(* Schneider Machine Expert - Basic project Seren_Alarm, file version 3.0.0.0 *)

HARDWARE
  Cpu 0: TM221CE16R
  EthernetConfiguration: NetworkName=M221, IpAllocationMode=FixedAddress, IpAddress=192.168.0.221, SubnetMask=255.255.255.0
  SerialLineConfiguration: Baud=Baud19200, Parity=ParityEven, DataBits=DataBits8, StopBits=StopBits1, PhysicalMedium=PhysicalMediumRs485, TransmissionMode=TransmissionModeModbusRtu, SlaveId=1, Addressing=SlaveAddressing
  MastTask: UsePeriodScanMode=false, PeriodScan=100
  FastTask: Period=255
  CpuBehavior: StartingMode=StartInRun, AutoSaveRamOnEeprom=true, WatchdogPeriod=250

SYMBOLS  (address, symbol, comment, settings)
  %M0       M_COM_OK
  %M1       M_HB_LAST
  %M2       M_HB_TOGGLED
  %M10      M_ENABLE_GEN
  %M11      M_PULSE_OUT
  %M12      M_PAUSE_OUT
  %M13      M_SERIES_PAUSE
  %S0       SB_COLDSTART  "Indicates or executes a cold start (data initialized to default values)"
  %MW0      PLC_CONTROL_WORD
  %MW1      PLC_STATUS_WORD
  %MW2      SOUND_PROFILE_CODE
  %MW3      SOUND_PULSE_COUNT
  %MW4      SOUND_PULSE_TIME_MS
  %MW5      SOUND_PAUSE_TIME_MS
  %MW6      SOUND_SERIES_INTERVAL_MS
  %MW10     ACTIVE_PULSE_COUNT
  %MW11     ACTIVE_PULSE_T_PRESET
  %MW12     ACTIVE_PAUSE_T_PRESET
  %MW13     ACTIVE_SERIES_T_PRESET
  %MW14     SERIES_COUNTER_VAL
  %TM0        [Preset=12, Base=OneSecond]
  %TM1        [Preset=2, Base=OneHundredMilliSeconds]
  %TM2        [Preset=3, Base=OneHundredMilliSeconds]
  %TM3        [Preset=30, Base=OneSecond]
  %QWM0     QW_HEARD_BEAT_WORD
  %QWM1     QW_PLC_CONTROL_WORD
  %IWM0     IW_PLC_HEARD_BEAT_WORD
  %IWM1     IW_PLC_STATUS_WORD

POU SIREN_CONTROL
  (* SectionNumber=1 *)

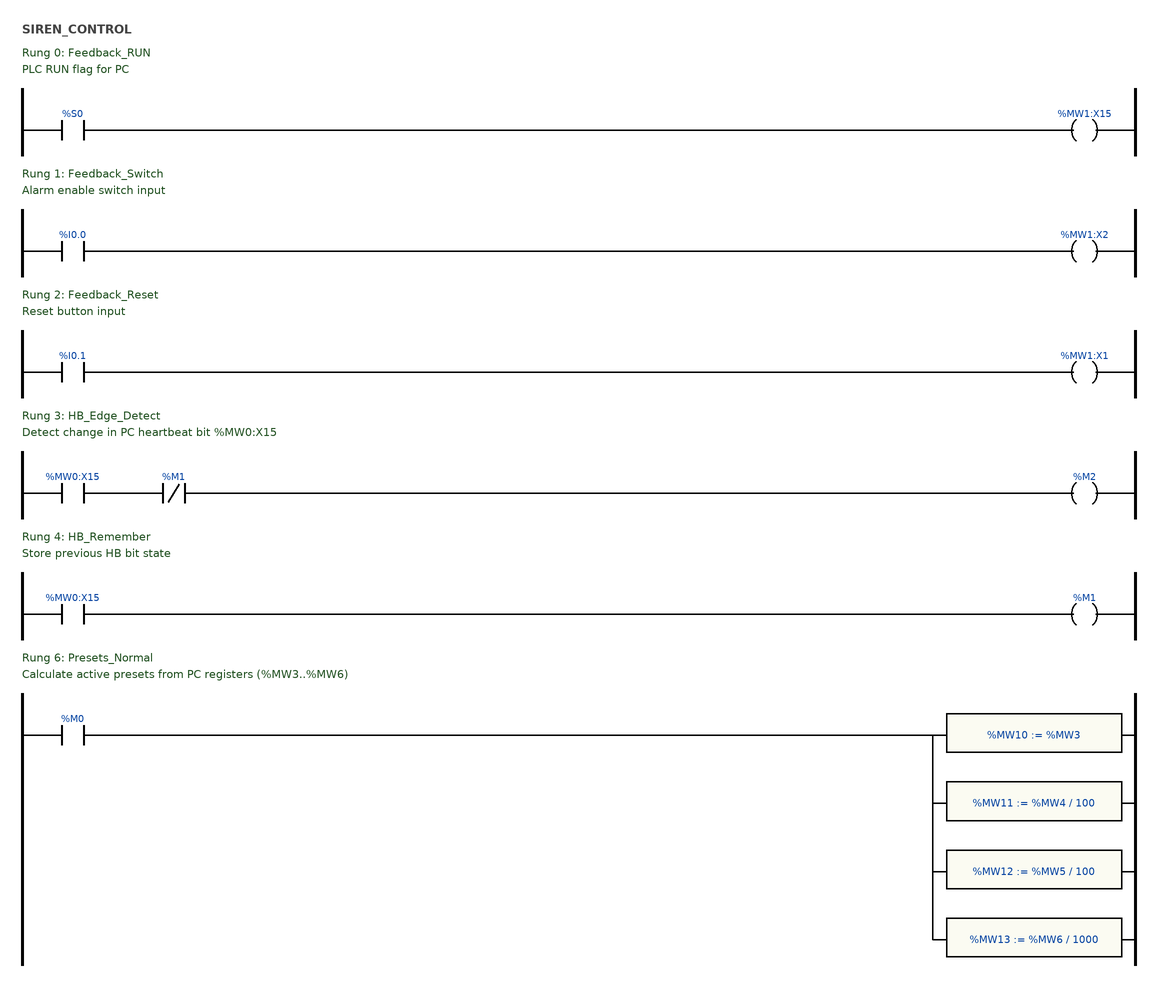

// Rung 0: Feedback_RUN
// PLC RUN flag for PC
  LD %S0                  (* SB_COLDSTART *)
  ST %MW1:X15             (* PLC_STATUS_WORD *)
  // as ST:
  //   PLC_STATUS_WORD:X15 := SB_COLDSTART;

// Rung 1: Feedback_Switch
// Alarm enable switch input
  LD %I0.0
  ST %MW1:X2              (* PLC_STATUS_WORD *)
  // as ST:
  //   PLC_STATUS_WORD:X2 := %I0.0;

// Rung 2: Feedback_Reset
// Reset button input
  LD %I0.1
  ST %MW1:X1              (* PLC_STATUS_WORD *)
  // as ST:
  //   PLC_STATUS_WORD:X1 := %I0.1;

// Rung 3: HB_Edge_Detect
// Detect change in PC heartbeat bit %MW0:X15
  LD %MW0:X15             (* PLC_CONTROL_WORD *)
  ANDN %M1                (* M_HB_LAST *)
  ST %M2                  (* M_HB_TOGGLED *)
  // as ST:
  //   M_HB_TOGGLED := PLC_CONTROL_WORD:X15 AND NOT M_HB_LAST;

// Rung 4: HB_Remember
// Store previous HB bit state
  LD %MW0:X15             (* PLC_CONTROL_WORD *)
  ST %M1                  (* M_HB_LAST *)
  // as ST:
  //   M_HB_LAST := PLC_CONTROL_WORD:X15;

// Rung 5: Watchdog_Timer
// Watchdog: %M0 is 1 while communication is OK, 0 when lost
  BLK %TM0
  LDN %M2                 (* M_HB_TOGGLED *)
  IN
  OUT_BLK
  LDN Q
  ST %M0                  (* M_COM_OK *)
  END_BLK
  // as ST:
  //   %TM0(IN := NOT M_HB_TOGGLED);
  //   M_COM_OK := NOT %TM0.Q;
  (* the ladder stored for this rung does not match its IL; not drawn *)

// Rung 6: Presets_Normal
// Calculate active presets from PC registers (%MW3..%MW6)
  LD %M0                  (* M_COM_OK *)
  [ %MW10 := %MW3 ]       (* ACTIVE_PULSE_COUNT, SOUND_PULSE_COUNT *)
  [ %MW11 := %MW4 / 100 ] (* ACTIVE_PULSE_T_PRESET, SOUND_PULSE_TIME_MS *)
  [ %MW12 := %MW5 / 100 ] (* ACTIVE_PAUSE_T_PRESET, SOUND_PAUSE_TIME_MS *)
  [ %MW13 := %MW6 / 1000 ](* ACTIVE_SERIES_T_PRESET, SOUND_SERIES_INTERVAL_MS *)
  // as ST:
  //   IF M_COM_OK THEN ACTIVE_PULSE_COUNT := SOUND_PULSE_COUNT; END_IF;
  //   IF M_COM_OK THEN ACTIVE_PULSE_T_PRESET := SOUND_PULSE_TIME_MS / 100; END_IF;
  //   IF M_COM_OK THEN ACTIVE_PAUSE_T_PRESET := SOUND_PAUSE_TIME_MS / 100; END_IF;
  //   IF M_COM_OK THEN ACTIVE_SERIES_T_PRESET := SOUND_SERIES_INTERVAL_MS / 1000; END_IF;

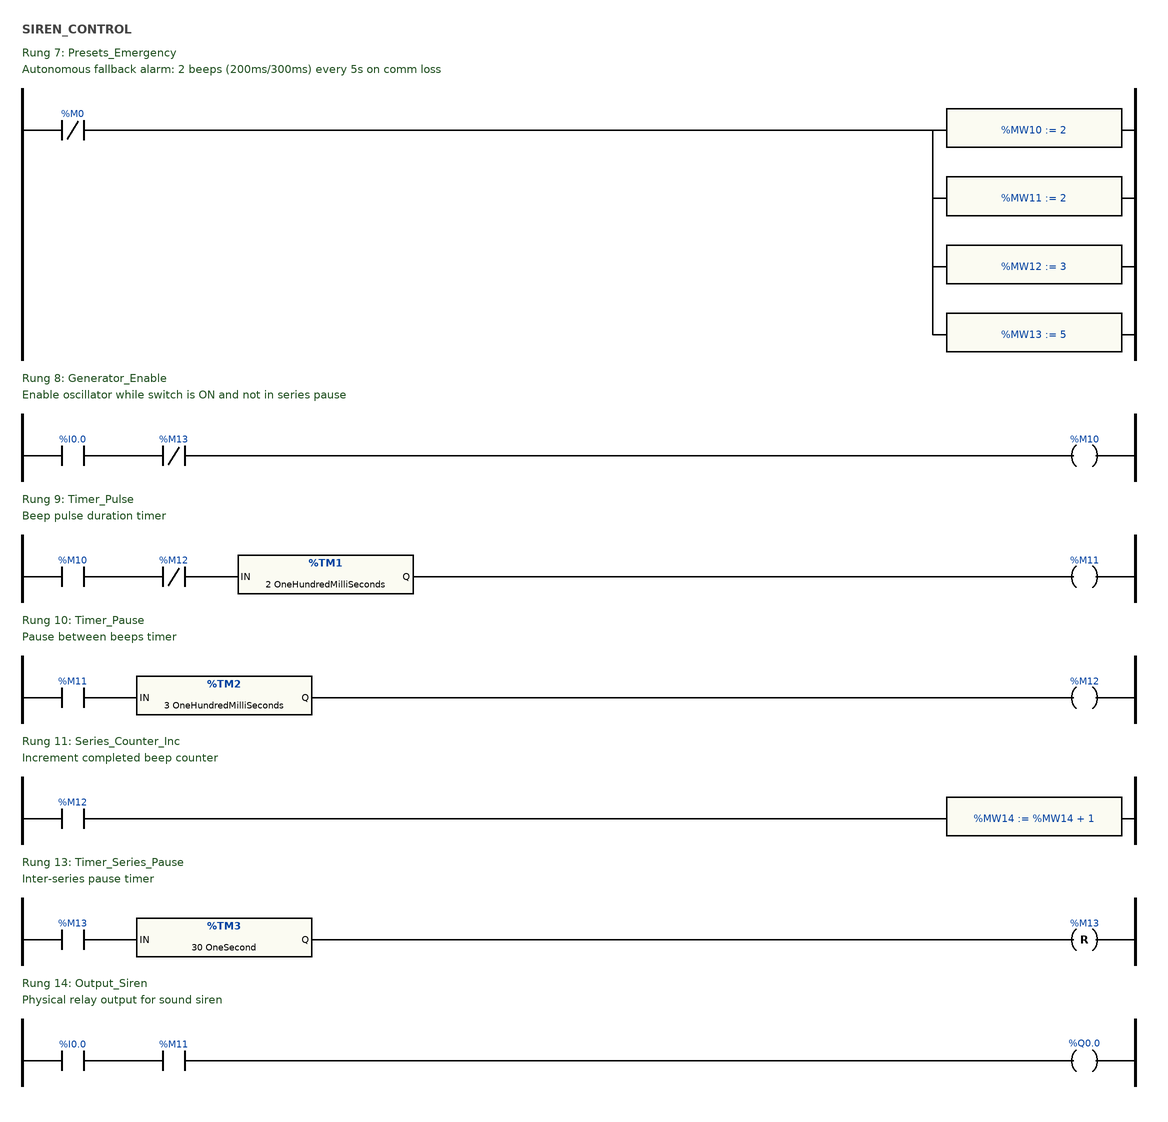

// Rung 7: Presets_Emergency
// Autonomous fallback alarm: 2 beeps (200ms/300ms) every 5s on comm loss
  LDN %M0                 (* M_COM_OK *)
  [ %MW10 := 2 ]          (* ACTIVE_PULSE_COUNT *)
  [ %MW11 := 2 ]          (* ACTIVE_PULSE_T_PRESET *)
  [ %MW12 := 3 ]          (* ACTIVE_PAUSE_T_PRESET *)
  [ %MW13 := 5 ]          (* ACTIVE_SERIES_T_PRESET *)
  // as ST:
  //   IF NOT M_COM_OK THEN ACTIVE_PULSE_COUNT := 2; END_IF;
  //   IF NOT M_COM_OK THEN ACTIVE_PULSE_T_PRESET := 2; END_IF;
  //   IF NOT M_COM_OK THEN ACTIVE_PAUSE_T_PRESET := 3; END_IF;
  //   IF NOT M_COM_OK THEN ACTIVE_SERIES_T_PRESET := 5; END_IF;

// Rung 8: Generator_Enable
// Enable oscillator while switch is ON and not in series pause
  LD %I0.0
  ANDN %M13               (* M_SERIES_PAUSE *)
  ST %M10                 (* M_ENABLE_GEN *)
  // as ST:
  //   M_ENABLE_GEN := %I0.0 AND NOT M_SERIES_PAUSE;

// Rung 9: Timer_Pulse
// Beep pulse duration timer
  BLK %TM1
  LD %M10                 (* M_ENABLE_GEN *)
  ANDN %M12               (* M_PAUSE_OUT *)
  IN
  OUT_BLK
  LD Q
  ST %M11                 (* M_PULSE_OUT *)
  END_BLK
  // as ST:
  //   %TM1(IN := M_ENABLE_GEN AND NOT M_PAUSE_OUT);
  //   M_PULSE_OUT := %TM1.Q;

// Rung 10: Timer_Pause
// Pause between beeps timer
  BLK %TM2
  LD %M11                 (* M_PULSE_OUT *)
  IN
  OUT_BLK
  LD Q
  ST %M12                 (* M_PAUSE_OUT *)
  END_BLK
  // as ST:
  //   %TM2(IN := M_PULSE_OUT);
  //   M_PAUSE_OUT := %TM2.Q;

// Rung 11: Series_Counter_Inc
// Increment completed beep counter
  LD %M12                 (* M_PAUSE_OUT *)
  [ %MW14 := %MW14 + 1 ]  (* SERIES_COUNTER_VAL, SERIES_COUNTER_VAL *)
  // as ST:
  //   IF M_PAUSE_OUT THEN SERIES_COUNTER_VAL := SERIES_COUNTER_VAL + 1; END_IF;

// Rung 12: Series_Finished
// Enter series pause when count reached
  LD %M10                 (* M_ENABLE_GEN *)
  AND [ %MW14 >= %MW10 ]  (* SERIES_COUNTER_VAL, ACTIVE_PULSE_COUNT *)
  S %M13                  (* M_SERIES_PAUSE *)
  [ %MW14 := 0 ]          (* SERIES_COUNTER_VAL *)
  // as ST:
  //   IF M_ENABLE_GEN AND SERIES_COUNTER_VAL >= ACTIVE_PULSE_COUNT THEN M_SERIES_PAUSE := TRUE; END_IF;
  //   IF M_ENABLE_GEN AND SERIES_COUNTER_VAL >= ACTIVE_PULSE_COUNT THEN SERIES_COUNTER_VAL := 0; END_IF;
  (* the ladder stored for this rung does not match its IL; not drawn *)

// Rung 13: Timer_Series_Pause
// Inter-series pause timer
  BLK %TM3
  LD %M13                 (* M_SERIES_PAUSE *)
  IN
  OUT_BLK
  LD Q
  R %M13                  (* M_SERIES_PAUSE *)
  END_BLK
  // as ST:
  //   %TM3(IN := M_SERIES_PAUSE);
  //   IF %TM3.Q THEN M_SERIES_PAUSE := FALSE; END_IF;

// Rung 14: Output_Siren
// Physical relay output for sound siren
  LD %I0.0
  AND %M11                (* M_PULSE_OUT *)
  ST %Q0.0
  // as ST:
  //   %Q0.0 := %I0.0 AND M_PULSE_OUT;

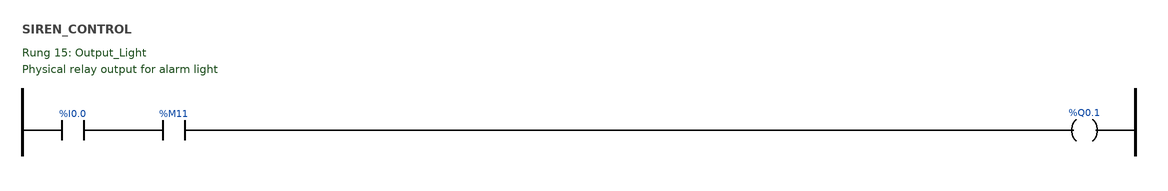

// Rung 15: Output_Light
// Physical relay output for alarm light
  LD %I0.0
  AND %M11                (* M_PULSE_OUT *)
  ST %Q0.1
  // as ST:
  //   %Q0.1 := %I0.0 AND M_PULSE_OUT;

POU ModBusExchange
  (* SectionNumber=2 *)

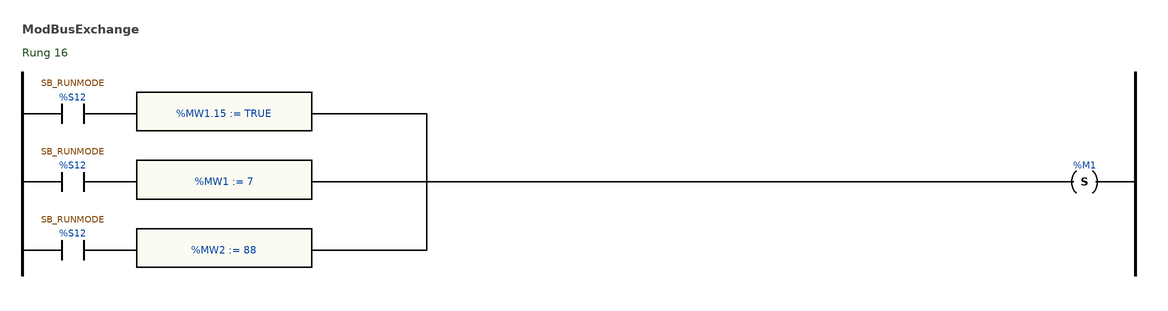

// Rung 16
  // %S12: The controller is running
  (* no IL stored for this rung *)
